FUNCTION_BLOCK INTERNAL FB_ValueDeviation_Tests EXTENDS FB_TestSuite
VAR_INPUT
END_VAR
VAR_OUTPUT
END_VAR
VAR
	_valueDeviation	: FB_ValueDeviation;
END_VAR

Test01_WhenDisabledStatusIsOk();
Test02_EnableWithNoDelay_ExpecteInstantError();
Test03_EnableWithDelay_ExpectErrorAfterDelayElapsed();
Test04_NoDelay_ChangeMaxDeviation_ExpectStatusAccordingToMaxValue();
Test05_StatusNOK_DisableAndExpectStatusOK();
Test06_NegativeMaxValue_ExpectTheDeviationAsAbsoluteValue();
Test07_NegativeValue();

METHOD PRIVATE Test01_WhenDisabledStatusIsOk
VAR_INPUT
END_VAR
TcUnit.TEST('Test01_WhenDisabledStatusIsOk');

_valueDeviation.Enable := FALSE;
_valueDeviation.MaxDeviation := 0;
_valueDeviation.Value.Setpoint := 100.0;
_valueDeviation.ActivationDelay := T#0S;
_valueDeviation();

AssertTrue(
	Condition := _valueDeviation.Status = E_ValueDeviationStatus.OK,
	Message := 'When disabled status should always be OK.');

TcUnit.TEST_FINISHED();
END_METHOD

METHOD Test02_EnableWithNoDelay_ExpecteInstantError
VAR_INPUT
END_VAR
TcUnit.TEST('Test02_EnableWithNoDelay_ExpecteInstantError');

_valueDeviation.Enable := TRUE;
_valueDeviation.MaxDeviation := 5;
_valueDeviation.ActivationDelay := T#0S;

_valueDeviation.Value.Setpoint := 10;
_valueDeviation.Value.Actual := 0;

_valueDeviation();

AssertTrue(
	Condition := _valueDeviation.Status = E_ValueDeviationStatus.NOK,
	Message := 'When enabled and no delay, status should be NOK when deviating over the threshold.');

_valueDeviation.Value.Setpoint := 10;
_valueDeviation.Value.Actual := 10;
_valueDeviation();

AssertTrue(
	Condition := _valueDeviation.Status = E_ValueDeviationStatus.OK,
	Message := 'When enabled and no delay, status should be OK when deviating under the threshold.');

TcUnit.TEST_FINISHED();
END_METHOD

METHOD Test03_EnableWithDelay_ExpectErrorAfterDelayElapsed : REFERENCE TO FB_Test
VAR_INPUT
END_VAR

VAR_INST
	TonDelayDeviation	: TON := (PT := T#1200MS);
	fbValueDeviation	: FB_ValueDeviation;
END_VAR
TcUnit.TEST('Test03_EnableWithDelay_ExpectErrorAfterDelayElapsed');

fbValueDeviation.Enable := TRUE;
fbValueDeviation.MaxDeviation := 0;
fbValueDeviation.Value.Setpoint := 100.0;
fbValueDeviation.Value.Actual := 50;
fbValueDeviation.ActivationDelay := T#1100MS;
fbValueDeviation();
TonDelayDeviation(IN := TRUE);

IF TonDelayDeviation.Q THEN
	AssertTrue(
	Condition := fbValueDeviation.Status = E_ValueDeviationStatus.NOK,
	Message := 'Deviation with delay after 1 second failed');

	TcUnit.TEST_FINISHED();
END_IF
END_METHOD

METHOD Test04_NoDelay_ChangeMaxDeviation_ExpectStatusAccordingToMaxValue
VAR_INPUT
END_VAR
TcUnit.TEST('Test04_NoDelay_ChangeMaxDeviation_ExpectStatusAccordingToMaxValue');

_valueDeviation.Enable := TRUE;
_valueDeviation.MaxDeviation := 100;
_valueDeviation.Value.Setpoint := 10;
_valueDeviation.Value.Actual := 2;
_valueDeviation.ActivationDelay := T#0S;
_valueDeviation();

AssertTrue(
	Condition := _valueDeviation.Status = E_ValueDeviationStatus.OK,
	Message := 'Changing threshold with no delay should instantly change status to OK when under max deviation.'
);

_valueDeviation.MaxDeviation := 5;
_valueDeviation();

AssertTrue(
	Condition := _valueDeviation.Status = E_ValueDeviationStatus.NOK,
	Message := 'Changing threshold with no delay should instantly change status to NOK when over max deviation.');

TcUnit.TEST_FINISHED();
END_METHOD

METHOD Test05_StatusNOK_DisableAndExpectStatusOK
VAR_INPUT
END_VAR
TcUnit.TEST('Test05_StatusNOK_DisableAndExpectStatusOK');

_valueDeviation.Enable := TRUE;
_valueDeviation.MaxDeviation := 0;
_valueDeviation.Value.Setpoint := 100.0;
_valueDeviation.Value.Actual := 500.0;
_valueDeviation.ActivationDelay := T#0S;
_valueDeviation();

AssertTrue(
	Condition := _valueDeviation.Status = E_ValueDeviationStatus.NOK,
	Message := 'Status should be NOK.'
);

_valueDeviation.Enable := FALSE;
_valueDeviation();

AssertTrue(
	Condition := _valueDeviation.Status = E_ValueDeviationStatus.OK,
	Message := 'When disabled status should always be OK.'
);

TcUnit.TEST_FINISHED();
END_METHOD

METHOD Test06_NegativeMaxValue_ExpectTheDeviationAsAbsoluteValue
VAR_INPUT
END_VAR
TcUnit.TEST('Test06_NegativeMaxValue_ExpectTheDeviationAsAbsoluteValue');

_valueDeviation.Enable := TRUE;
_valueDeviation.MaxDeviation := -10;
_valueDeviation.Value.Setpoint := 5;
_valueDeviation.Value.Actual := 8;
_valueDeviation.ActivationDelay := T#0S;
_valueDeviation();

AssertTrue(
	Condition := _valueDeviation.Status = E_ValueDeviationStatus.OK,
	Message := 'Expected status with set 5, act 8 and max deviation -10 is OK.');

_valueDeviation.MaxDeviation := -1;
_valueDeviation();

AssertTrue(
	Condition := _valueDeviation.Status = E_ValueDeviationStatus.NOK,
	Message := 'Expected status with set 5, act 8 and max deviation -1 is NOK.');


TcUnit.TEST_FINISHED();
END_METHOD

METHOD Test07_NegativeValue
VAR_INPUT
END_VAR
TcUnit.TEST('Test07_NegativeValue');

_valueDeviation.Enable := TRUE;
_valueDeviation.MaxDeviation := 10;
_valueDeviation.Value.Setpoint := -5;
_valueDeviation.Value.Actual := 0;
_valueDeviation.ActivationDelay := T#0S;
_valueDeviation();

AssertTrue(
	Condition := _valueDeviation.Status = E_ValueDeviationStatus.OK,
	Message := ' Expected status with set value -5, actual 0 and max deviation 10 is OK.');

_valueDeviation.Value.Setpoint := -15;
_valueDeviation();

AssertTrue(
	Condition := _valueDeviation.Status = E_ValueDeviationStatus.NOK,
	Message := 'Expected status with set value -15, actual 0 and max deviation 10 is NOK.');


TcUnit.TEST_FINISHED();
END_METHOD

END_FUNCTION_BLOCK

(* stored: Version 1.1.0.1, ProductVersion 3.1.4024.13
   POU FB_ValueDeviation_Tests: Id {23c2514e-c821-050c-065f-351b2b2d323f}, SpecialFunc None
   Method Test01_WhenDisabledStatusIsOk: Id {8818dded-160b-0207-259d-fc878542089b}
   Method Test02_EnableWithNoDelay_ExpecteInstantError: Id {4883a548-b068-0bad-0b31-7bb5a0136f22}
   Method Test03_EnableWithDelay_ExpectErrorAfterDelayElapsed: Id {3cd7c840-10f3-0ab2-1b51-6fbfe914e93a}
   Method Test04_NoDelay_ChangeMaxDeviation_ExpectStatusAccordingToMaxValue: Id {f948ae44-6cd3-07b9-340d-0ae066ad6ec4}
   Method Test05_StatusNOK_DisableAndExpectStatusOK: Id {5b5c1855-6eba-0dca-00e8-2f70bf539e4e}
   Method Test06_NegativeMaxValue_ExpectTheDeviationAsAbsoluteValue: Id {a54b0c5d-7bd5-0481-224c-5e05983eb7e5}
   Method Test07_NegativeValue: Id {47a55545-4e7f-062d-3b66-26c1f854476d} *)
